(* CODESYS project Automation-of-a-Production-Line-Codesys

Project tree, tasks and I/O mapping:
  Device : CODESYS Control Win V3 x64, 3S - Smart Software Solutions GmbH, version 3.5.18.30
    application Application
      libraries: Standard, 3.5.18.0 (System)
      task MainTask (cyclic, interval 35 ms, priority 1) calls Geral
      function block Enter_Piece_Up [SFC]
      program Geral [CFC]
      global variables GVL
      function block M3 [SFC]
      Symbols
      function block T_Lin_Double [SFC]
      function block T_Lin [SFC]
      function block T_Lin_Psh_Up [SFC]
      function block T_Rot_Down [SFC]
      function block T_Rot_Up [SFC]
      function block T_Transl_Down [SFC]
      function block T_Transl_Up [SFC]
      function block T_WH_in [SFC]: Enter_WH_exit
      function block T_WH_out [SFC]: Clear, Order
      program TimeMeas [ST]
      function block Tool_Counter [SFC]: Init_exit, Rot_Minus_exit, Rot_Plus_exit
    Ethernet : Ethernet, 3S - Smart Software Solutions GmbH, version 3.5.17.0
      Modbus_TCP_Master : Modbus TCP Master, 3S - Smart Software Solutions GmbH, version 4.2.0.0
          settings: AutoReconnect = TRUE
        Modbus_TCP_Slave : Modbus TCP Slave, 3S - Smart Software Solutions GmbH, version 4.1.0.0
            settings: Unit-ID = 255; ResponseTimeout = 100; IPAddress = [127, 0, 0, 1]; Port = 5502; Channel 0.Function Code = 2; Channel 0.Read Offset = 16#0000; Channel 0.Read Length = 99; Channel 0.Write Offset = 0; Channel 0.Write Length = 0; Channel 0.Cycle Time = 100; Channel 1.Function Code = 15; Channel 1.Read Offset = 0; Channel 1.Read Length = 0; Channel 1.Write Offset = 16#0000; Channel 1.Write Length = 126; Channel 1.Cycle Time = 100; Channel 2.Function Code = 16; Channel 2.Read Offset = 0; Channel 2.Read Length = 0; Channel 2.Write Offset = 16#0000; Channel 2.Write Length = 1; Channel 2.Cycle Time = 100
            input  Application.GVL.I[0] : BOOL  // Channel 0.Channel 0.Bit0
            input  Application.GVL.I[1] : BOOL  // Channel 0.Channel 0.Bit1
            input  Application.GVL.I[2] : BOOL  // Channel 0.Channel 0.Bit2
            input  Application.GVL.I[3] : BOOL  // Channel 0.Channel 0.Bit3
            input  Application.GVL.I[4] : BOOL  // Channel 0.Channel 0.Bit4
            input  Application.GVL.I[5] : BOOL  // Channel 0.Channel 0.Bit5
            input  Application.GVL.I[6] : BOOL  // Channel 0.Channel 0.Bit6
            input  Application.GVL.I[7] : BOOL  // Channel 0.Channel 0.Bit7
            input  Application.GVL.I[8] : BOOL  // Channel 0.Channel 0.Bit0
            input  Application.GVL.I[9] : BOOL  // Channel 0.Channel 0.Bit1
            input  Application.GVL.I[10] : BOOL  // Channel 0.Channel 0.Bit2
            input  Application.GVL.I[11] : BOOL  // Channel 0.Channel 0.Bit3
            input  Application.GVL.I[12] : BOOL  // Channel 0.Channel 0.Bit4
            input  Application.GVL.I[13] : BOOL  // Channel 0.Channel 0.Bit5
            input  Application.GVL.I[14] : BOOL  // Channel 0.Channel 0.Bit6
            input  Application.GVL.I[15] : BOOL  // Channel 0.Channel 0.Bit7
            input  Application.GVL.I[16] : BOOL  // Channel 0.Channel 0.Bit0
            input  Application.GVL.I[17] : BOOL  // Channel 0.Channel 0.Bit1
            input  Application.GVL.I[18] : BOOL  // Channel 0.Channel 0.Bit2
            input  Application.GVL.I[19] : BOOL  // Channel 0.Channel 0.Bit3
            input  Application.GVL.I[20] : BOOL  // Channel 0.Channel 0.Bit4
            input  Application.GVL.I[21] : BOOL  // Channel 0.Channel 0.Bit5
            input  Application.GVL.I[22] : BOOL  // Channel 0.Channel 0.Bit6
            input  Application.GVL.I[23] : BOOL  // Channel 0.Channel 0.Bit7
            input  Application.GVL.I[24] : BOOL  // Channel 0.Channel 0.Bit0
            input  Application.GVL.I[25] : BOOL  // Channel 0.Channel 0.Bit1
            input  Application.GVL.I[26] : BOOL  // Channel 0.Channel 0.Bit2
            input  Application.GVL.I[27] : BOOL  // Channel 0.Channel 0.Bit3
            input  Application.GVL.I[28] : BOOL  // Channel 0.Channel 0.Bit4
            input  Application.GVL.I[29] : BOOL  // Channel 0.Channel 0.Bit5
            input  Application.GVL.I[30] : BOOL  // Channel 0.Channel 0.Bit6
            input  Application.GVL.I[31] : BOOL  // Channel 0.Channel 0.Bit7
            input  Application.GVL.I[32] : BOOL  // Channel 0.Channel 0.Bit0
            input  Application.GVL.I[33] : BOOL  // Channel 0.Channel 0.Bit1
            input  Application.GVL.I[34] : BOOL  // Channel 0.Channel 0.Bit2
            input  Application.GVL.I[35] : BOOL  // Channel 0.Channel 0.Bit3
            input  Application.GVL.I[36] : BOOL  // Channel 0.Channel 0.Bit4
            input  Application.GVL.I[37] : BOOL  // Channel 0.Channel 0.Bit5
            input  Application.GVL.I[38] : BOOL  // Channel 0.Channel 0.Bit6
            input  Application.GVL.I[39] : BOOL  // Channel 0.Channel 0.Bit7
            input  Application.GVL.I[40] : BOOL  // Channel 0.Channel 0.Bit0
            input  Application.GVL.I[41] : BOOL  // Channel 0.Channel 0.Bit1
            input  Application.GVL.I[42] : BOOL  // Channel 0.Channel 0.Bit2
            input  Application.GVL.I[43] : BOOL  // Channel 0.Channel 0.Bit3
            input  Application.GVL.I[44] : BOOL  // Channel 0.Channel 0.Bit4
            input  Application.GVL.I[45] : BOOL  // Channel 0.Channel 0.Bit5
            input  Application.GVL.I[46] : BOOL  // Channel 0.Channel 0.Bit6
            input  Application.GVL.I[47] : BOOL  // Channel 0.Channel 0.Bit7
            input  Application.GVL.I[48] : BOOL  // Channel 0.Channel 0.Bit0
            input  Application.GVL.I[49] : BOOL  // Channel 0.Channel 0.Bit1
            input  Application.GVL.I[50] : BOOL  // Channel 0.Channel 0.Bit2
            input  Application.GVL.I[51] : BOOL  // Channel 0.Channel 0.Bit3
            input  Application.GVL.I[52] : BOOL  // Channel 0.Channel 0.Bit4
            input  Application.GVL.I[53] : BOOL  // Channel 0.Channel 0.Bit5
            input  Application.GVL.I[54] : BOOL  // Channel 0.Channel 0.Bit6
            input  Application.GVL.I[55] : BOOL  // Channel 0.Channel 0.Bit7
            input  Application.GVL.I[56] : BOOL  // Channel 0.Channel 0.Bit0
            input  Application.GVL.I[57] : BOOL  // Channel 0.Channel 0.Bit1
            input  Application.GVL.I[58] : BOOL  // Channel 0.Channel 0.Bit2
            input  Application.GVL.I[59] : BOOL  // Channel 0.Channel 0.Bit3
            input  Application.GVL.I[60] : BOOL  // Channel 0.Channel 0.Bit4
            input  Application.GVL.I[61] : BOOL  // Channel 0.Channel 0.Bit5
            input  Application.GVL.I[62] : BOOL  // Channel 0.Channel 0.Bit6
            input  Application.GVL.I[63] : BOOL  // Channel 0.Channel 0.Bit7
            input  Application.GVL.I[64] : BOOL  // Channel 0.Channel 0.Bit0
            input  Application.GVL.I[65] : BOOL  // Channel 0.Channel 0.Bit1
            input  Application.GVL.I[66] : BOOL  // Channel 0.Channel 0.Bit2
            input  Application.GVL.I[67] : BOOL  // Channel 0.Channel 0.Bit3
            input  Application.GVL.I[68] : BOOL  // Channel 0.Channel 0.Bit4
            input  Application.GVL.I[69] : BOOL  // Channel 0.Channel 0.Bit5
            input  Application.GVL.I[70] : BOOL  // Channel 0.Channel 0.Bit6
            input  Application.GVL.I[71] : BOOL  // Channel 0.Channel 0.Bit7
            input  Application.GVL.I[72] : BOOL  // Channel 0.Channel 0.Bit0
            input  Application.GVL.I[73] : BOOL  // Channel 0.Channel 0.Bit1
            input  Application.GVL.I[74] : BOOL  // Channel 0.Channel 0.Bit2
            input  Application.GVL.I[75] : BOOL  // Channel 0.Channel 0.Bit3
            input  Application.GVL.I[76] : BOOL  // Channel 0.Channel 0.Bit4
            input  Application.GVL.I[77] : BOOL  // Channel 0.Channel 0.Bit5
            input  Application.GVL.I[78] : BOOL  // Channel 0.Channel 0.Bit6
            input  Application.GVL.I[79] : BOOL  // Channel 0.Channel 0.Bit7
            input  Application.GVL.I[80] : BOOL  // Channel 0.Channel 0.Bit0
            input  Application.GVL.I[81] : BOOL  // Channel 0.Channel 0.Bit1
            input  Application.GVL.I[82] : BOOL  // Channel 0.Channel 0.Bit2
            input  Application.GVL.I[83] : BOOL  // Channel 0.Channel 0.Bit3
            input  Application.GVL.I[84] : BOOL  // Channel 0.Channel 0.Bit4
            input  Application.GVL.I[85] : BOOL  // Channel 0.Channel 0.Bit5
            input  Application.GVL.I[86] : BOOL  // Channel 0.Channel 0.Bit6
            input  Application.GVL.I[87] : BOOL  // Channel 0.Channel 0.Bit7
            input  Application.GVL.I[88] : BOOL  // Channel 0.Channel 0.Bit0
            input  Application.GVL.I[89] : BOOL  // Channel 0.Channel 0.Bit1
            input  Application.GVL.I[90] : BOOL  // Channel 0.Channel 0.Bit2
            input  Application.GVL.I[91] : BOOL  // Channel 0.Channel 0.Bit3
            input  Application.GVL.I[92] : BOOL  // Channel 0.Channel 0.Bit4
            input  Application.GVL.I[93] : BOOL  // Channel 0.Channel 0.Bit5
            input  Application.GVL.I[94] : BOOL  // Channel 0.Channel 0.Bit6
            input  Application.GVL.I[95] : BOOL  // Channel 0.Channel 0.Bit7
            input  Application.GVL.I[96] : BOOL  // Channel 0.Channel 0.Bit0
            input  Application.GVL.I[97] : BOOL  // Channel 0.Channel 0.Bit1
            input  Application.GVL.I[98] : BOOL  // Channel 0.Channel 0.Bit2
            output Application.GVL.O[0] : BOOL  // Channel 1.Channel 1.Bit0
            output Application.GVL.O[1] : BOOL  // Channel 1.Channel 1.Bit1
            output Application.GVL.O[2] : BOOL  // Channel 1.Channel 1.Bit2
            output Application.GVL.O[3] : BOOL  // Channel 1.Channel 1.Bit3
            output Application.GVL.O[4] : BOOL  // Channel 1.Channel 1.Bit4
            output Application.GVL.O[5] : BOOL  // Channel 1.Channel 1.Bit5
            output Application.GVL.O[6] : BOOL  // Channel 1.Channel 1.Bit6
            output Application.GVL.O[7] : BOOL  // Channel 1.Channel 1.Bit7
            output Application.GVL.O[8] : BOOL  // Channel 1.Channel 1.Bit0
            output Application.GVL.O[9] : BOOL  // Channel 1.Channel 1.Bit1
            output Application.GVL.O[10] : BOOL  // Channel 1.Channel 1.Bit2
            output Application.GVL.O[11] : BOOL  // Channel 1.Channel 1.Bit3
            output Application.GVL.O[12] : BOOL  // Channel 1.Channel 1.Bit4
            output Application.GVL.O[13] : BOOL  // Channel 1.Channel 1.Bit5
            output Application.GVL.O[14] : BOOL  // Channel 1.Channel 1.Bit6
            output Application.GVL.O[15] : BOOL  // Channel 1.Channel 1.Bit7
            output Application.GVL.O[16] : BOOL  // Channel 1.Channel 1.Bit0
            output Application.GVL.O[17] : BOOL  // Channel 1.Channel 1.Bit1
            output Application.GVL.O[18] : BOOL  // Channel 1.Channel 1.Bit2
            output Application.GVL.O[19] : BOOL  // Channel 1.Channel 1.Bit3
            output Application.GVL.O[20] : BOOL  // Channel 1.Channel 1.Bit4
            output Application.GVL.O[21] : BOOL  // Channel 1.Channel 1.Bit5
            output Application.GVL.O[22] : BOOL  // Channel 1.Channel 1.Bit6
            output Application.GVL.O[23] : BOOL  // Channel 1.Channel 1.Bit7
            output Application.GVL.O[24] : BOOL  // Channel 1.Channel 1.Bit0
            output Application.GVL.O[25] : BOOL  // Channel 1.Channel 1.Bit1
            output Application.GVL.O[26] : BOOL  // Channel 1.Channel 1.Bit2
            output Application.GVL.O[27] : BOOL  // Channel 1.Channel 1.Bit3
            output Application.GVL.O[28] : BOOL  // Channel 1.Channel 1.Bit4
            output Application.GVL.O[29] : BOOL  // Channel 1.Channel 1.Bit5
            output Application.GVL.O[30] : BOOL  // Channel 1.Channel 1.Bit6
            output Application.GVL.O[31] : BOOL  // Channel 1.Channel 1.Bit7
            output Application.GVL.O[32] : BOOL  // Channel 1.Channel 1.Bit0
            output Application.GVL.O[33] : BOOL  // Channel 1.Channel 1.Bit1
            output Application.GVL.O[34] : BOOL  // Channel 1.Channel 1.Bit2
            output Application.GVL.O[35] : BOOL  // Channel 1.Channel 1.Bit3
            output Application.GVL.O[36] : BOOL  // Channel 1.Channel 1.Bit4
            output Application.GVL.O[37] : BOOL  // Channel 1.Channel 1.Bit5
            output Application.GVL.O[38] : BOOL  // Channel 1.Channel 1.Bit6
            output Application.GVL.O[39] : BOOL  // Channel 1.Channel 1.Bit7
            output Application.GVL.O[40] : BOOL  // Channel 1.Channel 1.Bit0
            output Application.GVL.O[41] : BOOL  // Channel 1.Channel 1.Bit1
            output Application.GVL.O[42] : BOOL  // Channel 1.Channel 1.Bit2
            output Application.GVL.O[43] : BOOL  // Channel 1.Channel 1.Bit3
            output Application.GVL.O[44] : BOOL  // Channel 1.Channel 1.Bit4
            output Application.GVL.O[45] : BOOL  // Channel 1.Channel 1.Bit5
            output Application.GVL.O[46] : BOOL  // Channel 1.Channel 1.Bit6
            output Application.GVL.O[47] : BOOL  // Channel 1.Channel 1.Bit7
            output Application.GVL.O[48] : BOOL  // Channel 1.Channel 1.Bit0
            output Application.GVL.O[49] : BOOL  // Channel 1.Channel 1.Bit1
            output Application.GVL.O[50] : BOOL  // Channel 1.Channel 1.Bit2
            output Application.GVL.O[51] : BOOL  // Channel 1.Channel 1.Bit3
            output Application.GVL.O[52] : BOOL  // Channel 1.Channel 1.Bit4
            output Application.GVL.O[53] : BOOL  // Channel 1.Channel 1.Bit5
            output Application.GVL.O[54] : BOOL  // Channel 1.Channel 1.Bit6
            output Application.GVL.O[55] : BOOL  // Channel 1.Channel 1.Bit7
            output Application.GVL.O[56] : BOOL  // Channel 1.Channel 1.Bit0
            output Application.GVL.O[57] : BOOL  // Channel 1.Channel 1.Bit1
            output Application.GVL.O[58] : BOOL  // Channel 1.Channel 1.Bit2
            output Application.GVL.O[59] : BOOL  // Channel 1.Channel 1.Bit3
            output Application.GVL.O[60] : BOOL  // Channel 1.Channel 1.Bit4
            output Application.GVL.O[61] : BOOL  // Channel 1.Channel 1.Bit5
            output Application.GVL.O[62] : BOOL  // Channel 1.Channel 1.Bit6
            output Application.GVL.O[63] : BOOL  // Channel 1.Channel 1.Bit7
            output Application.GVL.O[64] : BOOL  // Channel 1.Channel 1.Bit0
            output Application.GVL.O[65] : BOOL  // Channel 1.Channel 1.Bit1
            output Application.GVL.O[66] : BOOL  // Channel 1.Channel 1.Bit2
            output Application.GVL.O[67] : BOOL  // Channel 1.Channel 1.Bit3
            output Application.GVL.O[68] : BOOL  // Channel 1.Channel 1.Bit4
            output Application.GVL.O[69] : BOOL  // Channel 1.Channel 1.Bit5
            output Application.GVL.O[70] : BOOL  // Channel 1.Channel 1.Bit6
            output Application.GVL.O[71] : BOOL  // Channel 1.Channel 1.Bit7
            output Application.GVL.O[72] : BOOL  // Channel 1.Channel 1.Bit0
            output Application.GVL.O[73] : BOOL  // Channel 1.Channel 1.Bit1
            output Application.GVL.O[74] : BOOL  // Channel 1.Channel 1.Bit2
            output Application.GVL.O[75] : BOOL  // Channel 1.Channel 1.Bit3
            output Application.GVL.O[76] : BOOL  // Channel 1.Channel 1.Bit4
            output Application.GVL.O[77] : BOOL  // Channel 1.Channel 1.Bit5
            output Application.GVL.O[78] : BOOL  // Channel 1.Channel 1.Bit6
            output Application.GVL.O[79] : BOOL  // Channel 1.Channel 1.Bit7
            output Application.GVL.O[80] : BOOL  // Channel 1.Channel 1.Bit0
            output Application.GVL.O[81] : BOOL  // Channel 1.Channel 1.Bit1
            output Application.GVL.O[82] : BOOL  // Channel 1.Channel 1.Bit2
            output Application.GVL.O[83] : BOOL  // Channel 1.Channel 1.Bit3
            output Application.GVL.O[84] : BOOL  // Channel 1.Channel 1.Bit4
            output Application.GVL.O[85] : BOOL  // Channel 1.Channel 1.Bit5
            output Application.GVL.O[86] : BOOL  // Channel 1.Channel 1.Bit6
            output Application.GVL.O[87] : BOOL  // Channel 1.Channel 1.Bit7
            output Application.GVL.O[88] : BOOL  // Channel 1.Channel 1.Bit0
            output Application.GVL.O[89] : BOOL  // Channel 1.Channel 1.Bit1
            output Application.GVL.O[90] : BOOL  // Channel 1.Channel 1.Bit2
            output Application.GVL.O[91] : BOOL  // Channel 1.Channel 1.Bit3
            output Application.GVL.O[92] : BOOL  // Channel 1.Channel 1.Bit4
            output Application.GVL.O[93] : BOOL  // Channel 1.Channel 1.Bit5
            output Application.GVL.O[94] : BOOL  // Channel 1.Channel 1.Bit6
            output Application.GVL.O[95] : BOOL  // Channel 1.Channel 1.Bit7
            output Application.GVL.O[96] : BOOL  // Channel 1.Channel 1.Bit0
            output Application.GVL.O[97] : BOOL  // Channel 1.Channel 1.Bit1
            output Application.GVL.O[98] : BOOL  // Channel 1.Channel 1.Bit2
            output Application.GVL.O[99] : BOOL  // Channel 1.Channel 1.Bit3
            output Application.GVL.O[100] : BOOL  // Channel 1.Channel 1.Bit4
            output Application.GVL.O[101] : BOOL  // Channel 1.Channel 1.Bit5
            output Application.GVL.O[102] : BOOL  // Channel 1.Channel 1.Bit6
            output Application.GVL.O[103] : BOOL  // Channel 1.Channel 1.Bit7
            output Application.GVL.O[104] : BOOL  // Channel 1.Channel 1.Bit0
            output Application.GVL.O[105] : BOOL  // Channel 1.Channel 1.Bit1
            output Application.GVL.O[106] : BOOL  // Channel 1.Channel 1.Bit2
            output Application.GVL.O[107] : BOOL  // Channel 1.Channel 1.Bit3
            output Application.GVL.O[108] : BOOL  // Channel 1.Channel 1.Bit4
            output Application.GVL.O[109] : BOOL  // Channel 1.Channel 1.Bit5
            output Application.GVL.O[110] : BOOL  // Channel 1.Channel 1.Bit6
            output Application.GVL.O[111] : BOOL  // Channel 1.Channel 1.Bit7
            output Application.GVL.O[112] : BOOL  // Channel 1.Channel 1.Bit0
            output Application.GVL.O[113] : BOOL  // Channel 1.Channel 1.Bit1
            output Application.GVL.O[114] : BOOL  // Channel 1.Channel 1.Bit2
            output Application.GVL.O[115] : BOOL  // Channel 1.Channel 1.Bit3
            output Application.GVL.O[116] : BOOL  // Channel 1.Channel 1.Bit4
            output Application.GVL.O[117] : BOOL  // Channel 1.Channel 1.Bit5
            output Application.GVL.O[118] : BOOL  // Channel 1.Channel 1.Bit6
            output Application.GVL.O[119] : BOOL  // Channel 1.Channel 1.Bit7
            output Application.GVL.O[120] : BOOL  // Channel 1.Channel 1.Bit0
            output Application.GVL.O[121] : BOOL  // Channel 1.Channel 1.Bit1
            output Application.GVL.O[122] : BOOL  // Channel 1.Channel 1.Bit2
            output Application.GVL.O[123] : BOOL  // Channel 1.Channel 1.Bit3
            output Application.GVL.O[124] : BOOL  // Channel 1.Channel 1.Bit4
            output Application.GVL.O[125] : BOOL  // Channel 1.Channel 1.Bit5
            output Application.GVL.R0 : WORD  // Channel 2.Channel 2
            unmapped channels: Channel 0, Channel 1, Channel 2
*)

// Device/Application/GVL
{attribute 'qualified_only'}
VAR_GLOBAL
	I : ARRAY [0..98] OF BOOL;
	O : ARRAY [0..125] OF BOOL;
	R0 : UINT;
END_VAR

// Device/Application/Geral
PROGRAM Geral
VAR
	WH_out: T_WH_out;
	T1: T_Lin;
	TR_Up_1: T_Rot_Up;
	T2: T_Lin;
	TR_Up_2: T_Rot_Up;
	TD: T_Lin_Double;
	TL1: T_Lin;
	TR_Up_3: T_Rot_Up;
	TL2: T_Lin;
	TR_Up_4: T_Rot_Up;
	TL3: T_Lin;
	Enter_Piece_Up0: Enter_Piece_Up;
	M3: M3;
	M4: M3;
	M1: M3;
	TL4: T_Lin;
	M2: M3;
	TL5: T_Lin;
	TL6: T_Lin;
	TD1: T_Lin_Double;
	TL7: T_Lin;
	TL8: T_Lin;
	Enter_Piece_Up1: Enter_Piece_Up;
	TL9: T_Lin;
	TD2: T_Lin_Double;
	TRD_1: T_Rot_Down;
	TRD_2: T_Rot_Down;
	TRD_3: T_Rot_Down;
	TRD_4: T_Rot_Down;
	TTUp: T_Transl_Up;
	TWH_in: T_WH_in;
	TLPsh_Up: T_Lin_Psh_Up;
	TLPsh_Up_D: T_Lin_Psh_Up;
	
	
	TTD: T_Transl_Down;
END_VAR
// Right -> MotorNeg
// Left -> MotorPos

TTD(
    sensor := GVL.I[44],
    free_M3_I := M3.free_O,
    recv_M4_I := M4.send_O,
    free_M4_I := M4.free_O,
    recv_M3_I := M3.send_O,
    free_V_I := TRD_2.free_O,
    recv_V_I := TRD_2.send_O,
    cmd_MR := TRUE,
    cmd_ML := FALSE,
    vertical := GVL.I[50],
    RIGHT_SIDE := GVL.I[45],
    LEFT_SIDE := GVL.I[46],
    cmd_R := TRUE,
    cmd_L := FALSE); // T_Transl_Down
GVL.O[67] := TTD.left;
GVL.O[68] := TTD.right;
GVL.O[69] := TTD.trans_left;
GVL.O[70] := TTD.trans_right;
T1(
    sensor := GVL.I[2],
    free_L_I := WH_out.free_O,
    free_R_I := TR_Up_1.free_O,
    recv_L_I := WH_out.send_O,
    recv_R_I := TR_Up_1.send_O,
    cmd_L := TRUE,
    cmd_R := FALSE); // T_Lin
WH_out(sensor := GVL.I[0], free_R_I := T1.free_O, cmd_R := TRUE, PieceToRemove := 5); // T_WH_out
GVL.O[5] := T1.left;
GVL.O[1] := WH_out.right;
GVL.O[6] := T1.right;
TR_Up_1(
    sensor := GVL.I[3],
    free_L_I := T1.free_O,
    free_R_I := T2.free_O,
    recv_L_I := T1.send_O,
    recv_R_I := T2.send_O,
    free_V_I := M1.free_O,
    recv_V_I := M1.send_O,
    cmd_L := TRUE,
    cmd_R := FALSE,
    cmd_Rotation_plus := FALSE,
    cmd_Rotation_minus := FALSE,
    horizontal := GVL.I[4],
    vertical := GVL.I[5]); // T_Rot_Up
GVL.O[7] := TR_Up_1.left;
GVL.O[8] := TR_Up_1.right;
GVL.O[10] := TR_Up_1.rotate_plus;
GVL.O[9] := TR_Up_1.rotate_minus;
T2(
    sensor := GVL.I[23],
    free_L_I := TR_Up_1.free_O,
    free_R_I := TR_Up_2.free_O,
    recv_L_I := TR_Up_1.send_O,
    recv_R_I := TR_Up_2.send_O,
    cmd_L := TRUE,
    cmd_R := FALSE); // T_Lin
GVL.O[37] := T2.left;
GVL.O[38] := T2.right;
TR_Up_2(
    sensor := GVL.I[24],
    free_L_I := T2.free_O,
    free_R_I := TD.free_O,
    recv_L_I := T2.send_O,
    recv_R_I := TD.send_O,
    free_V_I := TTUp.free_O,
    recv_V_I := TTUp.send_O,
    cmd_L := TRUE,
    cmd_R := FALSE,
    cmd_Rotation_plus := FALSE,
    cmd_Rotation_minus := FALSE,
    horizontal := GVL.I[25],
    vertical := GVL.I[26]); // T_Rot_Up
GVL.O[42] := TR_Up_2.rotate_plus;
GVL.O[41] := TR_Up_2.rotate_minus;
GVL.O[40] := TR_Up_2.right;
GVL.O[39] := TR_Up_2.left;
TD(
    sensor_left := GVL.I[27],
    sensor_right := GVL.I[28],
    free_L_I := TR_Up_2.free_O,
    free_R_I := TL1.free_O,
    recv_L_I := TR_Up_2.send_O,
    recv_R_I := TL1.send_O,
    cmd_L := TRUE,
    cmd_R := FALSE); // T_Lin_Double
GVL.O[43] := TD.left;
GVL.O[44] := TD.right;
TL1(
    sensor := GVL.I[53],
    free_L_I := TD.free_O,
    free_R_I := TR_Up_3.free_O,
    recv_L_I := TD.send_O,
    recv_R_I := TR_Up_3.send_O,
    cmd_L := TRUE,
    cmd_R := FALSE); // T_Lin
GVL.O[79] := TL1.left;
GVL.O[80] := TL1.right;
TR_Up_3(
    sensor := GVL.I[54],
    free_L_I := TL1.free_O,
    free_R_I := TL2.free_O,
    recv_L_I := TL1.send_O,
    recv_R_I := TL2.send_O,
    free_V_I := TD2.free_O,
    recv_V_I := TD2.send_O,
    cmd_L := TRUE,
    cmd_R := FALSE,
    cmd_Rotation_plus := FALSE,
    cmd_Rotation_minus := FALSE,
    horizontal := GVL.I[25],
    vertical := GVL.I[26]); // T_Rot_Up
GVL.O[81] := TR_Up_3.left;
GVL.O[82] := TR_Up_3.right;
GVL.O[83] := TR_Up_3.rotate_plus;
GVL.O[84] := TR_Up_3.rotate_minus;
TL2(
    sensor := GVL.I[77],
    free_L_I := TR_Up_3.free_O,
    free_R_I := TR_Up_4.free_O,
    recv_L_I := TR_Up_3.send_O,
    recv_R_I := TR_Up_4.send_O,
    cmd_L := TRUE,
    cmd_R := FALSE); // T_Lin
GVL.O[102] := TL2.left;
GVL.O[103] := TL2.right;
TR_Up_4(
    sensor := GVL.I[78],
    free_L_I := TL2.free_O,
    free_R_I := Enter_Piece_Up0.free_O,
    recv_L_I := TL2.send_O,
    recv_R_I := Enter_Piece_Up0.send_O,
    free_V_I := FALSE,
    recv_V_I := FALSE,
    cmd_L := TRUE,
    cmd_R := FALSE,
    cmd_Rotation_plus := FALSE,
    cmd_Rotation_minus := FALSE,
    horizontal := GVL.I[79],
    vertical := GVL.I[80]); // T_Rot_Up
GVL.O[104] := TR_Up_4.left;
Enter_Piece_Up0(sensor := GVL.I[81], free_L_I := TR_Up_4.free_O, recv_L_I := TR_Up_4.send_O, cmd_L := TRUE); // Enter_Piece_Up
GVL.O[105] := TR_Up_4.right;
GVL.O[107] := TR_Up_4.rotate_minus;
GVL.O[108] := Enter_Piece_Up0.left;
GVL.O[106] := TR_Up_4.rotate_plus;
M4(
    sensor := GVL.I[38],
    free_L_I := TTUp.free_O,
    free_R_I := TTD.free_O,
    recv_L_I := TTUp.send_O,
    recv_R_I := TTD.send_O,
    cmd_L := FALSE,
    cmd_R := TRUE,
    tool_ready := GVL.I[39],
    cmd_R_plus := FALSE,
    cmd_R_minus := FALSE,
    cmd_stop := T#20s,
    cmd_run := TRUE); // M3
GVL.O[58] := M4.left;
GVL.O[59] := M4.right;
GVL.O[62] := M4.Producing;
GVL.O[60] := M4.plus;
GVL.O[61] := M4.minus;
TD2(
    sensor_left := GVL.I[57],
    sensor_right := GVL.I[58],
    free_L_I := TR_Up_3.free_O,
    free_R_I := TL9.free_O,
    recv_L_I := TR_Up_3.send_O,
    recv_R_I := TL9.send_O,
    cmd_L := FALSE,
    cmd_R := TRUE); // T_Lin_Double
GVL.O[86] := TD2.right;
GVL.O[85] := TD2.left;
TL9(
    sensor := GVL.I[59],
    free_L_I := TD2.free_O,
    free_R_I := TRD_3.free_O,
    recv_L_I := TD2.send_O,
    recv_R_I := TRD_3.send_O,
    cmd_L := FALSE,
    cmd_R := TRUE); // T_Lin
GVL.O[87] := TL9.left;
GVL.O[88] := TL9.right;
TTUp(
    sensor := GVL.I[29],
    free_M3_I := M3.free_O,
    recv_M4_I := M4.free_O,
    free_M4_I := M4.send_O,
    recv_M3_I := M3.send_O,
    free_V_I := TR_Up_2.free_O,
    recv_V_I := TR_Up_2.send_O,
    cmd_MR := TRUE,
    cmd_ML := FALSE,
    vertical := GVL.I[26],
    RIGHT_SIDE := GVL.I[31],
    LEFT_SIDE := GVL.I[30],
    cmd_R := TRUE,
    cmd_L := FALSE); // T_Transl_Up
GVL.O[45] := TTUp.left;
GVL.O[46] := TTUp.right;
GVL.O[47] := TTUp.trans_left;
GVL.O[48] := TTUp.trans_right;
M3(
    sensor := GVL.I[32],
    free_L_I := TTUp.free_O,
    free_R_I := TTD.free_O,
    recv_L_I := TTUp.send_O,
    recv_R_I := TTD.send_O,
    cmd_L := FALSE,
    cmd_R := TRUE,
    tool_ready := GVL.I[32],
    cmd_R_plus := FALSE,
    cmd_R_minus := FALSE,
    cmd_stop := T#20s,
    cmd_run := TRUE);
GVL.O[53] := M3.Producing;
GVL.O[49] := M3.left;
GVL.O[50] := M3.right;
GVL.O[51] := M3.plus;
GVL.O[52] := M3.minus;
M1(
    sensor := GVL.I[6],
    free_L_I := TR_Up_1.free_O,
    free_R_I := TL4.free_O,
    recv_L_I := TR_Up_1.send_O,
    recv_R_I := TL4.send_O,
    cmd_L := TRUE,
    cmd_R := FALSE,
    tool_ready := GVL.I[7],
    cmd_R_plus := FALSE,
    cmd_R_minus := FALSE,
    cmd_stop := T#20s,
    cmd_run := TRUE); // M3
GVL.O[11] := M1.left;
GVL.O[12] := M1.right;
GVL.O[13] := M1.plus;
GVL.O[14] := M1.minus;
GVL.O[15] := M1.Producing;
TL4(
    sensor := GVL.I[12],
    free_L_I := M1.free_O,
    free_R_I := M2.free_O,
    recv_L_I := M1.send_O,
    recv_R_I := M2.send_O,
    cmd_L := FALSE,
    cmd_R := TRUE); // T_Lin
GVL.O[21] := TL4.right;
GVL.O[20] := TL4.left;
M2(
    sensor := GVL.I[13],
    free_L_I := TL4.free_O,
    free_R_I := TRD_1.free_O,
    recv_L_I := TL4.send_O,
    recv_R_I := TRD_1.send_O,
    cmd_L := TRUE,
    cmd_R := FALSE,
    tool_ready := GVL.I[14],
    cmd_R_plus := FALSE,
    cmd_R_minus := FALSE,
    cmd_stop := T#20s,
    cmd_run := TRUE); // M3
GVL.O[26] := M2.Producing;
GVL.O[24] := M2.plus;
GVL.O[25] := M2.minus;
GVL.O[22] := M2.left;
GVL.O[23] := M2.right;
TLPsh_Up(
    sensor := GVL.I[82],
    free_L_I := TR_Up_4.free_O,
    free_R_I := TLPsh_Up_D.free_O,
    recv_L_I := TR_Up_4.send_O,
    recv_R_I := TLPsh_Up_D.send_O,
    cmd_L := FALSE,
    cmd_R := FALSE,
    cmd_in := TRUE,
    contracted := GVL.I[83],
    extended := GVL.I[84],
    space_free := GVL.I[93]); // T_Lin_Psh_Up
GVL.O[113] := TLPsh_Up.transl_R;
GVL.O[110] := TLPsh_Up.left;
GVL.O[112] := TLPsh_Up.transl_L;
GVL.O[111] := TLPsh_Up.right;
TLPsh_Up_D(
    sensor := GVL.I[85],
    free_L_I := TLPsh_Up.free_O,
    free_R_I := TRD_4.free_O,
    recv_L_I := TLPsh_Up.send_O,
    recv_R_I := TRD_4.send_O,
    cmd_L := TRUE,
    cmd_R := FALSE,
    cmd_in := FALSE,
    contracted := GVL.I[86],
    extended := GVL.I[87],
    space_free := GVL.I[94]); // T_Lin_Psh_Up
GVL.O[114] := TLPsh_Up_D.left;
GVL.O[115] := TLPsh_Up_D.right;
GVL.O[117] := TLPsh_Up_D.transl_R;
GVL.O[116] := TLPsh_Up_D.transl_L;
TWH_in(
    sensor := GVL.I[1],
    free_R_I := TL5.free_O,
    recv_R_I := TL5.send_O,
    free_L_I := TRUE,
    cmd_R := FALSE,
    cmd_L := TRUE); // T_WH_in
GVL.O[3] := TWH_in.right;
GVL.O[2] := TWH_in.left;
GVL.O[4] := TWH_in.IN;
TL5(
    sensor := GVL.I[22],
    free_L_I := TWH_in.free_O,
    free_R_I := TRD_1.free_O,
    recv_L_I := TWH_in.send_O,
    recv_R_I := TRD_1.send_O,
    cmd_L := TRUE,
    cmd_R := FALSE); // T_Lin
GVL.O[35] := TL5.left;
GVL.O[36] := TL5.right;
TRD_1(
    sensor := GVL.I[19],
    free_L_I := TL5.free_O,
    free_R_I := TL6.free_O,
    recv_L_I := TL5.send_O,
    recv_R_I := TL6.send_O,
    free_V_I := M2.free_O,
    recv_V_I := M2.send_O,
    cmd_L := TRUE,
    cmd_R := FALSE,
    cmd_Rotation_plus := FALSE,
    cmd_Rotation_minus := FALSE,
    horizontal := GVL.I[20],
    vertical := GVL.I[21]); // T_Rot_Down
GVL.O[31] := TRD_1.left;
GVL.O[32] := TRD_1.right;
GVL.O[33] := TRD_1.rotate_plus;
GVL.O[34] := TRD_1.rotate_minus;
TL6(
    sensor := GVL.I[47],
    free_L_I := TRD_1.free_O,
    free_R_I := TRD_2.free_O,
    recv_L_I := TRD_1.send_O,
    recv_R_I := TRD_2.send_O,
    cmd_L := TRUE,
    cmd_R := FALSE); // T_Lin
GVL.O[71] := TL6.left;
GVL.O[72] := TL6.right;
TRD_2(
    sensor := GVL.I[48],
    free_L_I := TL6.free_O,
    free_R_I := TD1.free_O,
    recv_L_I := TL6.send_O,
    recv_R_I := TD1.send_O,
    free_V_I := TTD.free_O,
    recv_V_I := TTD.send_O,
    cmd_L := TRUE,
    cmd_R := FALSE,
    cmd_Rotation_plus := FALSE,
    cmd_Rotation_minus := FALSE,
    horizontal := GVL.I[49],
    vertical := GVL.I[50]); // T_Rot_Down
GVL.O[73] := TRD_2.left;
GVL.O[74] := TRD_2.right;
GVL.O[75] := TRD_2.rotate_plus;
GVL.O[76] := TRD_2.rotate_minus;
TD1(
    sensor_left := GVL.I[51],
    sensor_right := GVL.I[52],
    free_L_I := TRD_2.free_O,
    free_R_I := TL7.free_O,
    recv_L_I := TRD_2.send_O,
    recv_R_I := TL7.send_O,
    cmd_L := TRUE,
    cmd_R := FALSE); // T_Lin_Double
GVL.O[77] := TD1.left;
GVL.O[78] := TD1.right;
TL7(
    sensor := GVL.I[60],
    free_L_I := TD1.free_O,
    free_R_I := TRD_3.free_O,
    recv_L_I := TD1.send_O,
    recv_R_I := TRD_3.send_O,
    cmd_L := TRUE,
    cmd_R := FALSE); // T_Lin
GVL.O[89] := TL7.left;
GVL.O[90] := TL7.right;
TRD_3(
    sensor := GVL.I[61],
    free_L_I := TL7.free_O,
    free_R_I := TL8.free_O,
    recv_L_I := TL7.send_O,
    recv_R_I := TL8.send_O,
    free_V_I := TL9.free_O,
    recv_V_I := TL9.send_O,
    cmd_L := TRUE,
    cmd_R := FALSE,
    cmd_Rotation_plus := FALSE,
    cmd_Rotation_minus := FALSE,
    horizontal := GVL.I[62],
    vertical := GVL.I[63]); // T_Rot_Down
GVL.O[91] := TRD_3.left;
GVL.O[92] := TRD_3.right;
GVL.O[93] := TRD_3.rotate_plus;
GVL.O[94] := TRD_3.rotate_minus;
TL8(
    sensor := GVL.I[88],
    free_L_I := TRD_3.free_O,
    free_R_I := TRD_4.free_O,
    recv_L_I := TRD_3.send_O,
    recv_R_I := TRD_4.send_O,
    cmd_L := TRUE,
    cmd_R := FALSE); // T_Lin
GVL.O[118] := TL8.left;
GVL.O[119] := TL8.right;
TRD_4(
    sensor := GVL.I[89],
    free_L_I := TL8.free_O,
    free_R_I := Enter_Piece_Up1.free_O,
    recv_L_I := TL8.send_O,
    recv_R_I := Enter_Piece_Up1.send_O,
    free_V_I := TLPsh_Up_D.free_O,
    recv_V_I := TLPsh_Up_D.send_O,
    cmd_L := TRUE,
    cmd_R := FALSE,
    cmd_Rotation_plus := FALSE,
    cmd_Rotation_minus := FALSE,
    horizontal := GVL.I[90],
    vertical := GVL.I[91]); // T_Rot_Down
Enter_Piece_Up1(sensor := GVL.I[92], free_L_I := TRD_4.free_O, recv_L_I := TRD_4.send_O, cmd_L := TRUE); // Enter_Piece_Up
GVL.O[120] := TRD_4.left;
GVL.O[121] := TRD_4.right;
GVL.O[122] := TRD_4.rotate_plus;
GVL.O[124] := Enter_Piece_Up1.left;
GVL.O[125] := Enter_Piece_Up1.right;
GVL.O[123] := TRD_4.rotate_minus;

END_PROGRAM

// Device/Application/T_Lin_Double
FUNCTION_BLOCK T_Lin_Double
VAR_INPUT
	sensor_left: BOOL;
	sensor_right: BOOL;
	free_L_I: BOOL;
	free_R_I: BOOL;
	recv_L_I: BOOL;
	recv_R_I: BOOL;
	cmd_L:BOOL;
	cmd_R:BOOL;
		
END_VAR
VAR_OUTPUT
	left : BOOL;
	right : BOOL;
	free_O: BOOL;
	send_O: BOOL;
END_VAR
VAR
END_VAR

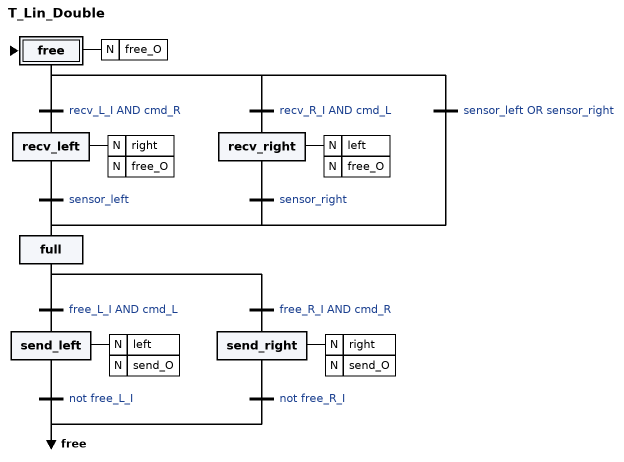
INITIAL_STEP free:
    free_O(N);
END_STEP
TRANSITION FROM free TO recv_left
    := recv_L_I AND cmd_R;
END_TRANSITION
STEP recv_left:
    right(N);
    free_O(N);
END_STEP
TRANSITION FROM recv_left TO full
    := sensor_left;
END_TRANSITION
TRANSITION FROM free TO recv_right
    := recv_R_I AND cmd_L;
END_TRANSITION
STEP recv_right:
    left(N);
    free_O(N);
END_STEP
TRANSITION FROM recv_right TO full
    := sensor_right;
END_TRANSITION
TRANSITION FROM free TO full
    := sensor_left OR sensor_right;
END_TRANSITION
STEP full:
END_STEP
TRANSITION FROM full TO send_left
    := free_L_I AND cmd_L;
END_TRANSITION
STEP send_left:
    left(N);
    send_O(N);
END_STEP
TRANSITION FROM send_left TO free
    := not free_L_I;
END_TRANSITION
TRANSITION FROM full TO send_right
    := free_R_I AND cmd_R;
END_TRANSITION
STEP send_right:
    right(N);
    send_O(N);
END_STEP
TRANSITION FROM send_right TO free
    := not free_R_I;
END_TRANSITION

END_FUNCTION_BLOCK

// Device/Application/Enter_Piece_Up
FUNCTION_BLOCK Enter_Piece_Up
VAR_INPUT
	sensor: BOOL;
	free_L_I: BOOL;
	recv_L_I: BOOL;
	cmd_L:BOOL;
	cmd_R: BOOL;
			
END_VAR
VAR_OUTPUT
	left : BOOL;
	right : BOOL;
	free_O: BOOL;
	send_O: BOOL;
END_VAR
VAR
END_VAR

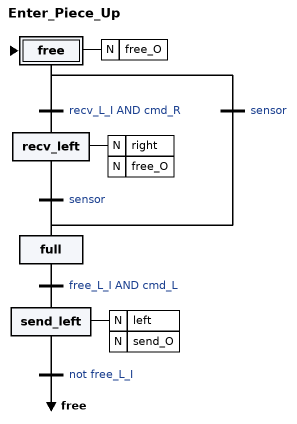
INITIAL_STEP free:
    free_O(N);
END_STEP
TRANSITION FROM free TO recv_left
    := recv_L_I AND cmd_R;
END_TRANSITION
STEP recv_left:
    right(N);
    free_O(N);
END_STEP
TRANSITION FROM recv_left TO full
    := sensor;
END_TRANSITION
TRANSITION FROM free TO full
    := sensor;
END_TRANSITION
STEP full:
END_STEP
TRANSITION FROM full TO send_left
    := free_L_I AND cmd_L;
END_TRANSITION
STEP send_left:
    left(N);
    send_O(N);
END_STEP
TRANSITION FROM send_left TO free
    := not free_L_I;
END_TRANSITION

END_FUNCTION_BLOCK

// Device/Application/T_Rot_Up
FUNCTION_BLOCK T_Rot_Up
VAR_INPUT
	sensor: BOOL;
	free_L_I: BOOL;
	free_R_I: BOOL;
	recv_L_I: BOOL;
	recv_R_I: BOOL;
	free_V_I: BOOL;
	recv_V_I: BOOL;
	cmd_L:BOOL;
	cmd_R:BOOL;
	cmd_Rotation_plus: BOOL;
	cmd_Rotation_minus: BOOL;
	horizontal: BOOL;
	vertical: BOOL;
	
END_VAR
VAR_OUTPUT
	left : BOOL;
	right : BOOL;
	rotate_plus : BOOL;
	rotate_minus : BOOL;
	free_O: BOOL;
	send_O: BOOL;
END_VAR
VAR
END_VAR

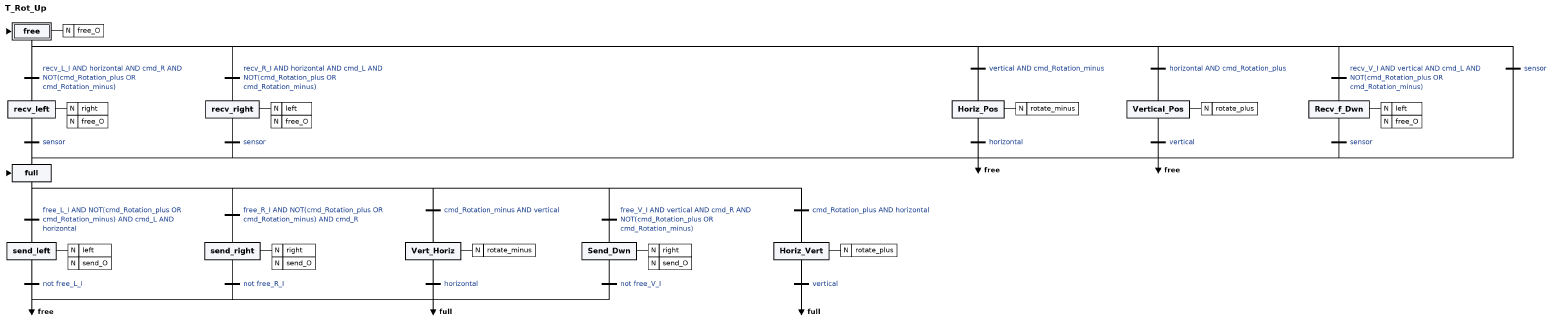
INITIAL_STEP free:
    free_O(N);
END_STEP
TRANSITION FROM free TO recv_left
    := recv_L_I AND horizontal AND cmd_R AND NOT(cmd_Rotation_plus OR cmd_Rotation_minus);
END_TRANSITION
STEP recv_left:
    right(N);
    free_O(N);
END_STEP
TRANSITION FROM recv_left TO full
    := sensor;
END_TRANSITION
TRANSITION FROM free TO recv_right
    := recv_R_I AND horizontal AND cmd_L AND NOT(cmd_Rotation_plus OR cmd_Rotation_minus);
END_TRANSITION
STEP recv_right:
    left(N);
    free_O(N);
END_STEP
TRANSITION FROM recv_right TO full
    := sensor;
END_TRANSITION
TRANSITION FROM free TO Horiz_Pos
    := vertical AND cmd_Rotation_minus;
END_TRANSITION
STEP Horiz_Pos:
    rotate_minus(N);
END_STEP
TRANSITION FROM Horiz_Pos TO free
    := horizontal;
END_TRANSITION
TRANSITION FROM free TO Vertical_Pos
    := horizontal AND cmd_Rotation_plus;
END_TRANSITION
STEP Vertical_Pos:
    rotate_plus(N);
END_STEP
TRANSITION FROM Vertical_Pos TO free
    := vertical;
END_TRANSITION
TRANSITION FROM free TO Recv_f_Dwn
    := recv_V_I AND vertical AND cmd_L AND NOT(cmd_Rotation_plus OR cmd_Rotation_minus);
END_TRANSITION
STEP Recv_f_Dwn:
    left(N);
    free_O(N);
END_STEP
TRANSITION FROM Recv_f_Dwn TO full
    := sensor;
END_TRANSITION
TRANSITION FROM free TO full
    := sensor;
END_TRANSITION
STEP full:
END_STEP
TRANSITION FROM full TO send_left
    := free_L_I AND NOT(cmd_Rotation_plus OR cmd_Rotation_minus) AND cmd_L AND horizontal;
END_TRANSITION
STEP send_left:
    left(N);
    send_O(N);
END_STEP
TRANSITION FROM send_left TO free
    := not free_L_I;
END_TRANSITION
TRANSITION FROM full TO send_right
    := free_R_I AND NOT(cmd_Rotation_plus OR cmd_Rotation_minus) AND cmd_R;
END_TRANSITION
STEP send_right:
    right(N);
    send_O(N);
END_STEP
TRANSITION FROM send_right TO free
    := not free_R_I;
END_TRANSITION
TRANSITION FROM full TO Vert_Horiz
    := cmd_Rotation_minus AND vertical;
END_TRANSITION
STEP Vert_Horiz:
    rotate_minus(N);
END_STEP
TRANSITION FROM Vert_Horiz TO full
    := horizontal;
END_TRANSITION
TRANSITION FROM full TO Send_Dwn
    := free_V_I AND vertical AND cmd_R AND NOT(cmd_Rotation_plus OR cmd_Rotation_minus);
END_TRANSITION
STEP Send_Dwn:
    right(N);
    send_O(N);
END_STEP
TRANSITION FROM Send_Dwn TO free
    := not free_V_I;
END_TRANSITION
TRANSITION FROM full TO Horiz_Vert
    := cmd_Rotation_plus AND horizontal;
END_TRANSITION
STEP Horiz_Vert:
    rotate_plus(N);
END_STEP
TRANSITION FROM Horiz_Vert TO full
    := vertical;
END_TRANSITION

END_FUNCTION_BLOCK

// Device/Application/T_Lin
FUNCTION_BLOCK T_Lin
VAR_INPUT
	sensor: BOOL;
	free_L_I: BOOL;
	free_R_I: BOOL;
	recv_L_I: BOOL;
	recv_R_I: BOOL;
	cmd_L:BOOL;
	cmd_R:BOOL;
		
END_VAR
VAR_OUTPUT
	left : BOOL;
	right : BOOL;
	free_O: BOOL;
	send_O: BOOL;
END_VAR
VAR
END_VAR

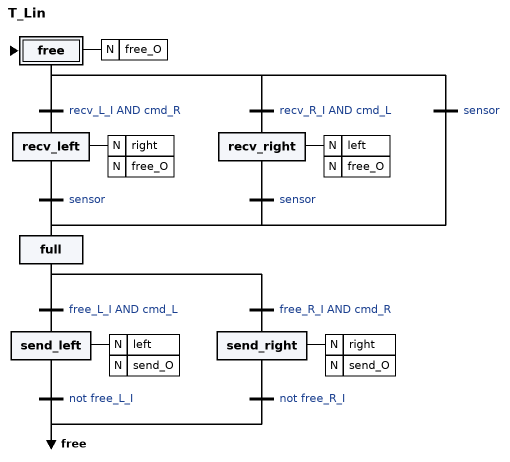
INITIAL_STEP free:
    free_O(N);
END_STEP
TRANSITION FROM free TO recv_left
    := recv_L_I AND cmd_R;
END_TRANSITION
STEP recv_left:
    right(N);
    free_O(N);
END_STEP
TRANSITION FROM recv_left TO full
    := sensor;
END_TRANSITION
TRANSITION FROM free TO recv_right
    := recv_R_I AND cmd_L;
END_TRANSITION
STEP recv_right:
    left(N);
    free_O(N);
END_STEP
TRANSITION FROM recv_right TO full
    := sensor;
END_TRANSITION
TRANSITION FROM free TO full
    := sensor;
END_TRANSITION
STEP full:
END_STEP
TRANSITION FROM full TO send_left
    := free_L_I AND cmd_L;
END_TRANSITION
STEP send_left:
    left(N);
    send_O(N);
END_STEP
TRANSITION FROM send_left TO free
    := not free_L_I;
END_TRANSITION
TRANSITION FROM full TO send_right
    := free_R_I AND cmd_R;
END_TRANSITION
STEP send_right:
    right(N);
    send_O(N);
END_STEP
TRANSITION FROM send_right TO free
    := not free_R_I;
END_TRANSITION

END_FUNCTION_BLOCK

// Device/Application/M3
FUNCTION_BLOCK M3
VAR_INPUT
	sensor: BOOL;
	free_L_I: BOOL;
	free_R_I: BOOL;
	recv_L_I: BOOL;
	recv_R_I: BOOL;
	cmd_L:BOOL;
	cmd_R:BOOL;
	tool_ready: BOOL;
	cmd_R_plus: BOOL;
	cmd_R_minus: BOOL;
	cmd_stop: TIME;
	cmd_run: BOOL;
	
		
END_VAR
VAR_OUTPUT
	left : BOOL;
	right : BOOL;
	free_O: BOOL;
	send_O: BOOL;
	plus: BOOL;
	minus: BOOL;
	Producing: BOOL;
END_VAR
VAR
		
END_VAR

